Fanuc KAREL source: ka00055.KL

-- PROVISIONAL review KL for V770-1; original PC SHA256 313cc04c07c7f84ff0969d9267a9290a1eb4c91d0864aeb682f5cfbf229fe25e
-- Incomplete behavior may be omitted. Consult companion uncertainty JSON. Do not deploy.
PROGRAM KA00055
%NOLOCKGROUP
-- UNRESOLVED_DECL SRC type=000101
-- UNRESOLVED_DECL DST type=000106
BEGIN
  -- UNRESOLVED_PC offsets 5-25; opcodes 49,7E,4A
  -- UNRESOLVED_PC offsets 30-34; opcodes 7F
END KA00055
